PROGRAM MAIN
VAR 
{attribute 'OPC.UA.DA' := '1'}
    hi:BOOL;
    timer: ton;
	{attribute 'OPC.UA.DA' := '1'}
	FIO_Input : BOOL;
{attribute 'OPC.UA.DA' := '1'}
	FIO_Output : BOOL; 
	testbit: BOOL;
END_VAR

// U; Pupu
// PW: 1

(*SUUNNITELMA
Vain pari structia missä on {attribute} päällä eli menee opc:lle jakoon
Niiden alle keräis jollain logiikalla kaikki jaettavat muuttujat.
	Simuloiden tilannetta missä asiakkaalle pitäisi se jakaa
	"tärkeät" asiat eli merkityksellinen data
	Toiminnallinen data
Laitekohtaisesti ryhmitelty? 
Erikseen vielä in/out ryhmä missä tietoa vois vaihtaa HMI:lle tms

PART 2
Toteutetaan hiukan OOP tai POP -tyyliä -> Vähennetään GVL käyttöä
Sagatowskin "PLC programming using TwinCAT 3 - Function blocks & interfaces (Part 6a/18)" video
	On käytössä valmista koodia mitä jokatapauksessa tulee muokattua niin voi heitellä ympäriinsä ja järjestellä mieluisaksi
	
*)

testbit := FIO_Output;

timer(IN := NOT timer.Q, PT := T#1S) ;
IF timer.Q THEN
    hi := NOT hi;
	FIO_Input := NOT FIO_Input;
END_IF

END_PROGRAM

(* stored: Version 1.1.0.1, ProductVersion 3.1.4024.12
   POU MAIN: Id {27056a27-a1e6-4813-a15f-14bfb1b953a1}, SpecialFunc None *)
